// TIA Portal V19 export
DATA_BLOCK "CYCLE_POPUP"   // DB37
{ S7_Optimized_Access := 'FALSE' }
   VAR
      "RINSE-1_START_YES" : Bool;
      "RINSE-1_START_NO" : Bool;
      "RINSE-1_RECIRCULATION" : Bool;
      "RINSE-1_DRAIN" : Bool;
      "RINSE-2_START_YES" : Bool;
      "RINSE-2_START_NO" : Bool;
      "RINSE-2_RECIRCULATION" : Bool;
      "RINSE-2_DRAIN" : Bool;
      "ACID/ALKALI_START_YES" : Bool;
      "ACID/ALKALI_START_NO" : Bool;
      "ALKALI/ACID_RECIRCULATION" : Bool;
      "ALKALI/ACID_DRAIN" : Bool;
      "ACID/ALKALI CONTINUE CYCLE" : Bool;
      "RINSE-3_START_YES" : Bool;
      "RINSE-3_START_NO" : Bool;
      "RINSE-3_RECIRCULATION" : Bool;
      "RINSE-3_DRAIN" : Bool;
      FINAL_RINSE_START_YES : Bool;
      FINAL_RINSE_START_NO : Bool;
      FINAL_RINSE_RECIRCULATION : Bool;
      FINAL_RINSE_FRESH_CYCLE : Bool;
      ALKALI : Bool;
      ACID : Bool;
      "ALKALI /ACID FRESH CYCLE" : Bool;
      FINAL_RINSE_DRAIN : Bool;
      "SW TANK_START_YES" : Bool;
      "SW TANK_START_NO" : Bool;
      "PW TANK_START_YES" : Bool;
      "PW TANK_START_NO" : Bool;
      "PW TANK_START_YES1" : Bool;
   END_VAR
BEGIN
END_DATA_BLOCK
